// TIA Portal V20 export
FUNCTION "E001" : Void   // FC2, FBD
{ S7_Optimized_Access := 'TRUE' }
// stored: SetENOAutomatically false
   VAR_TEMP
      Stirrer_TimeMs : DInt;
      State : "Service_States";
   END_VAR
BEGIN

REGION Network 1: Channel input
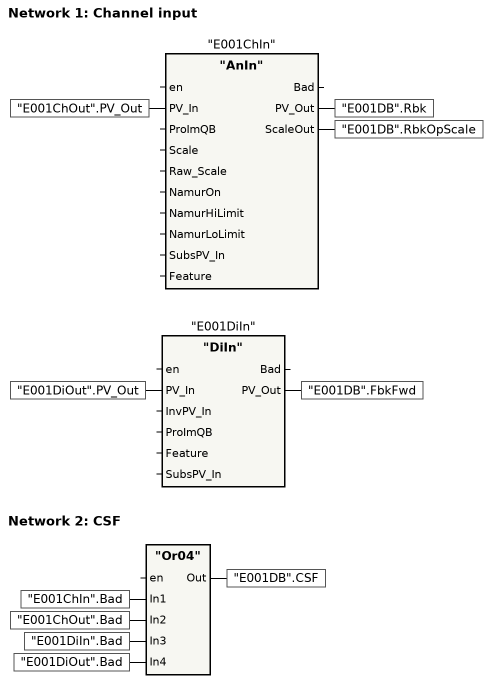
   "E001ChIn"(PV_In := "E001ChOut".PV_Out, PV_Out => "E001DB".Rbk, ScaleOut => "E001DB".RbkOpScale);   // "AnIn"
   "E001DiIn"(PV_In := "E001DiOut".PV_Out, PV_Out => "E001DB".FbkFwd);   // "DiIn"
END_REGION

REGION Network 2: CSF
   "Or04"(In1 := "E001ChIn".Bad,
          In2 := "E001ChOut".Bad,
          In3 := "E001DiIn".Bad,
          In4 := "E001DiOut".Bad,
          Out => "E001DB".CSF);
END_REGION

REGION Network 3: Interlock
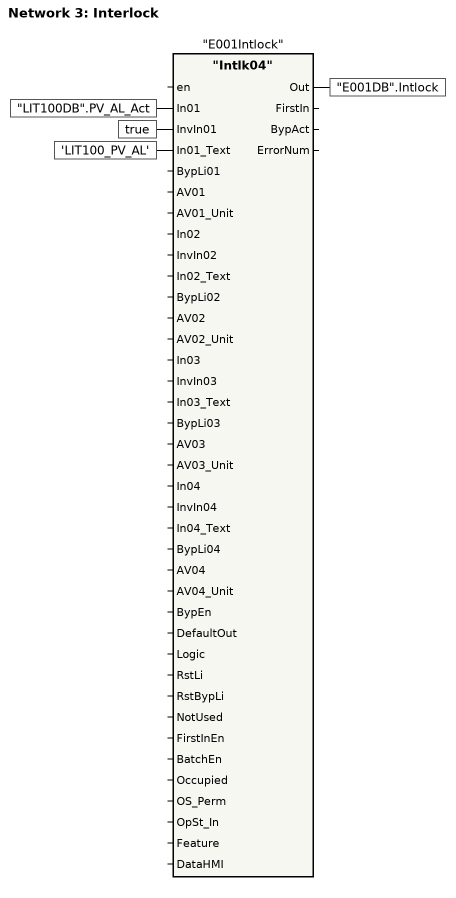
   "E001Intlock"(In01 := "LIT100DB".PV_AL_Act,   // "Intlk04"
                 InvIn01 := true,
                 In01_Text := 'LIT100_PV_AL',
                 Out => "E001DB".Intlock);
END_REGION

REGION Network 4: MotSpdCL
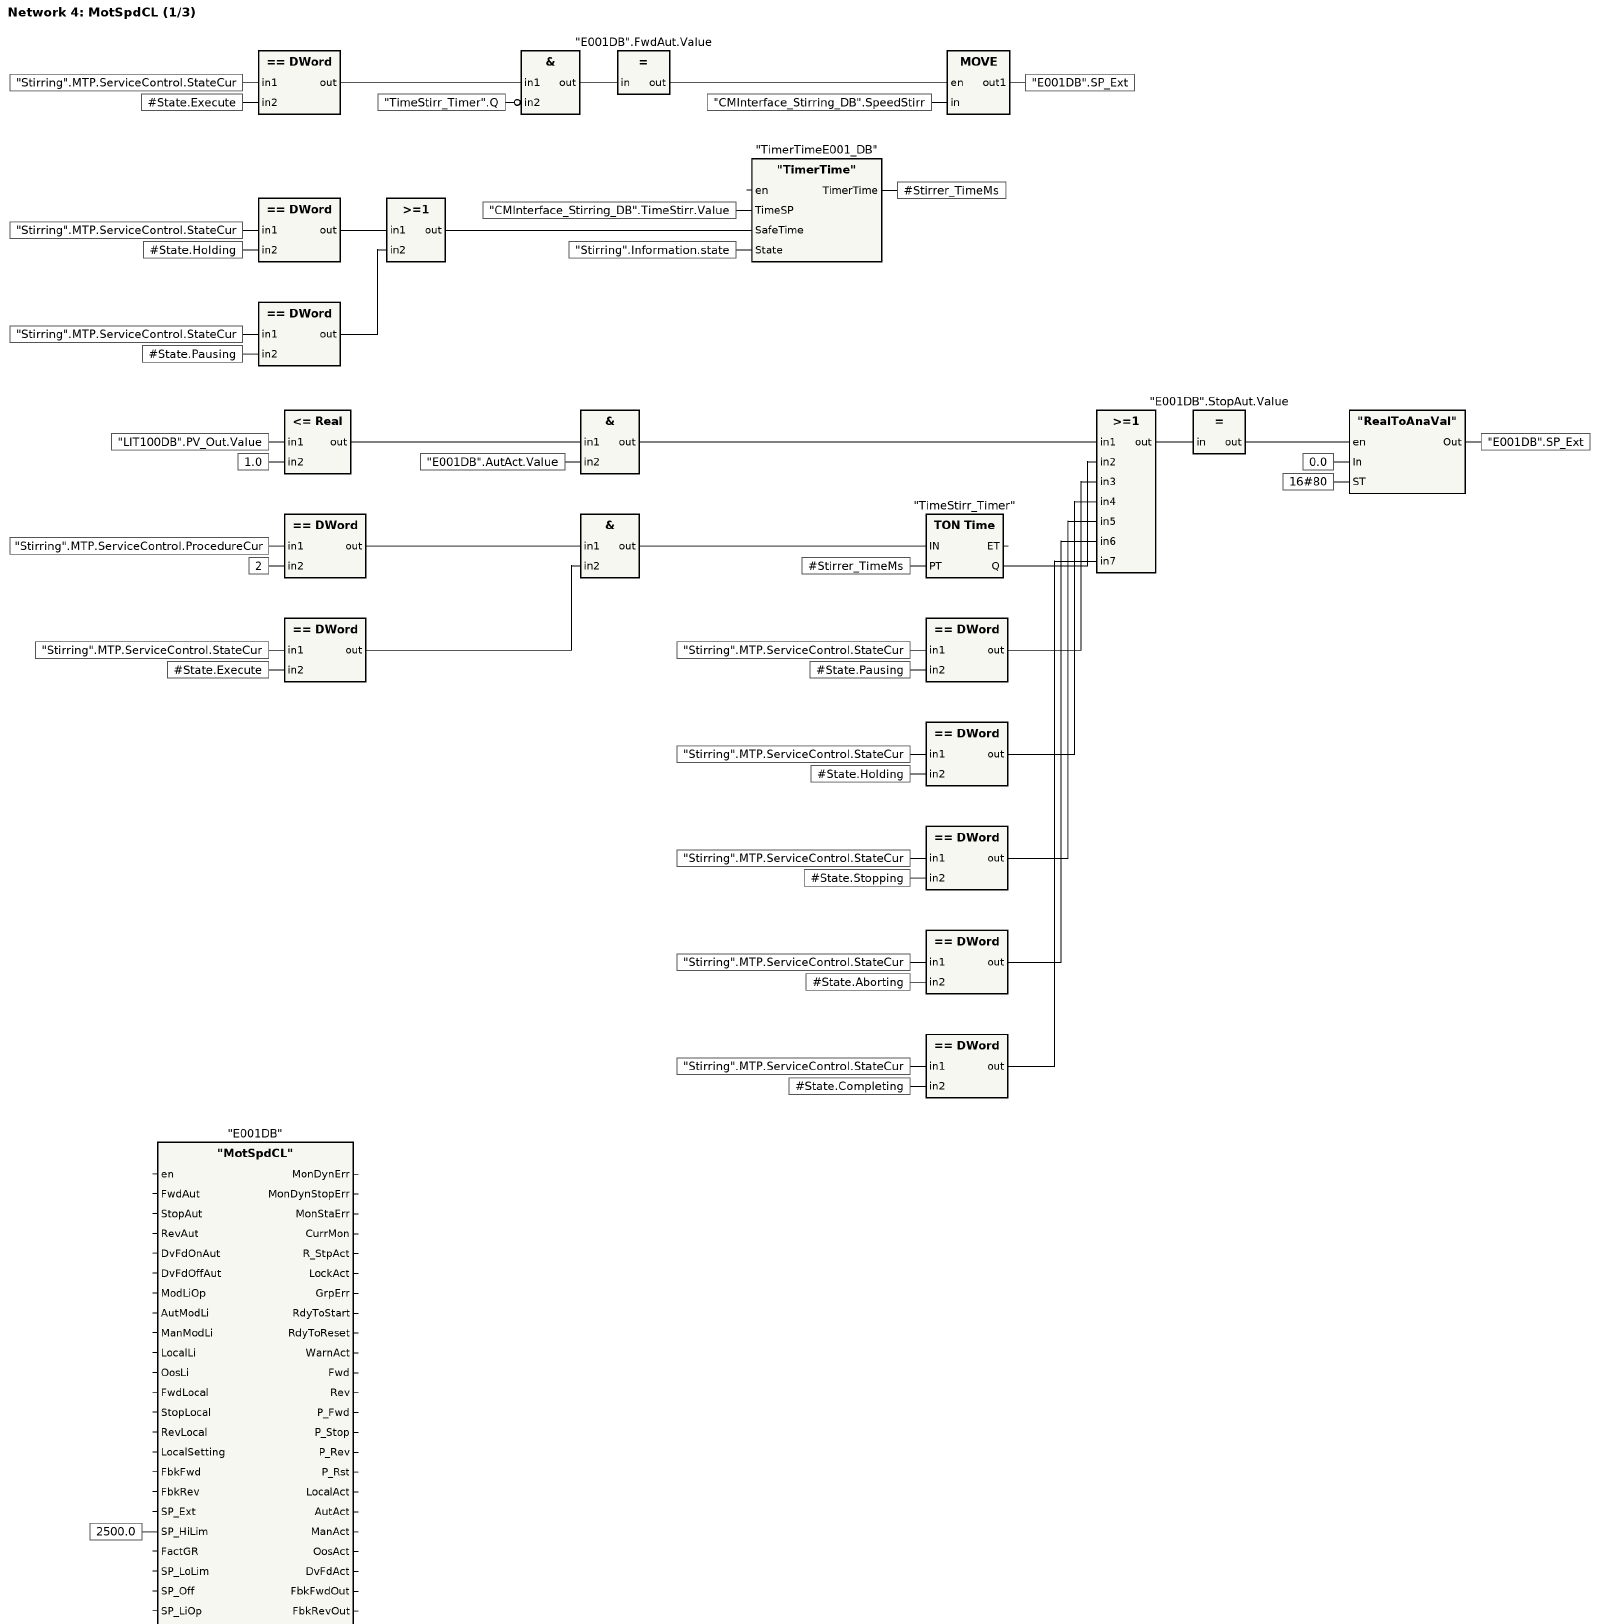
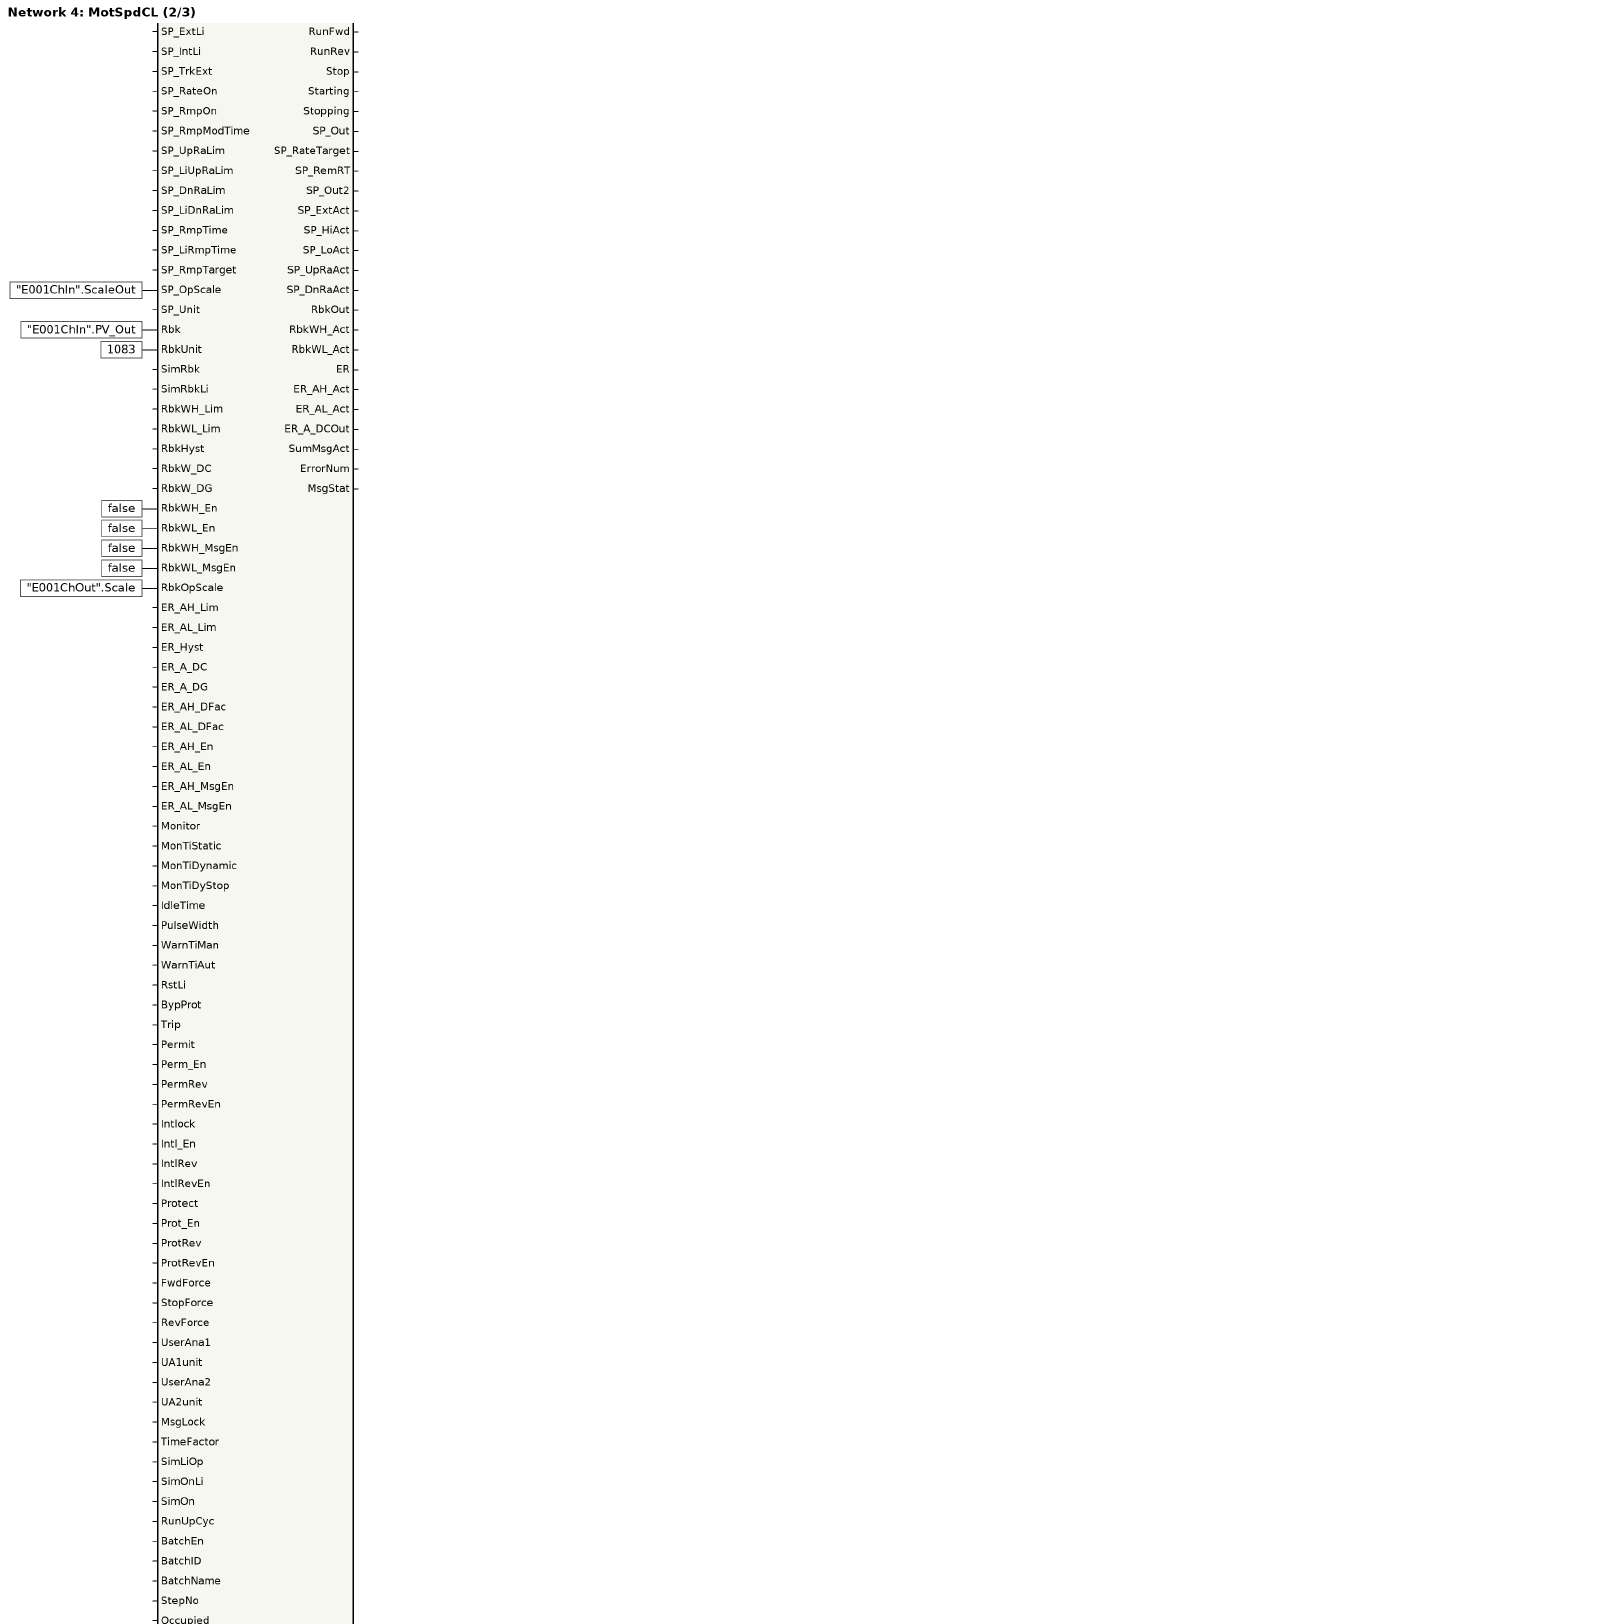
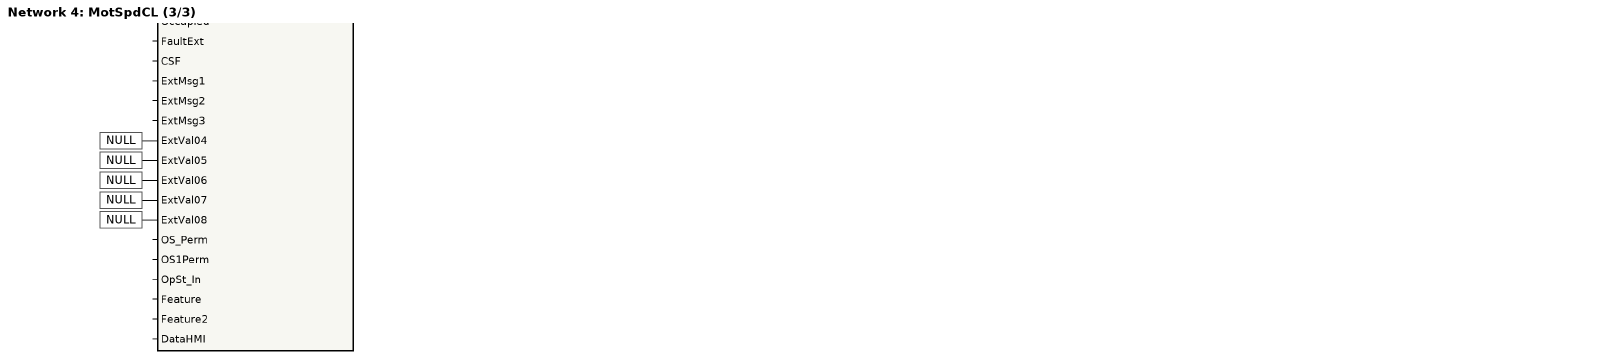
   "E001DB".FwdAut.Value := ("Stirring".MTP.ServiceControl.StateCur = #State.Execute) AND NOT "TimeStirr_Timer".Q;
   IF "E001DB".FwdAut.Value THEN "E001DB".SP_Ext := "CMInterface_Stirring_DB".SpeedStirr; END_IF;
   "TimerTimeE001_DB"(TimeSP := "CMInterface_Stirring_DB".TimeStirr.Value,   // "TimerTime"
                      SafeTime := ("Stirring".MTP.ServiceControl.StateCur = #State.Holding) OR ("Stirring".MTP.ServiceControl.StateCur = #State.Pausing),
                      State := "Stirring".Information.state,
                      TimerTime => #Stirrer_TimeMs);
   "TimeStirr_Timer".TON(IN := ("Stirring".MTP.ServiceControl.ProcedureCur = 2) AND ("Stirring".MTP.ServiceControl.StateCur = #State.Execute),
                         PT := #Stirrer_TimeMs);
   "E001DB".StopAut.Value := (("LIT100DB".PV_Out.Value <= 1.0) AND "E001DB".AutAct.Value) OR "TimeStirr_Timer".Q OR ("Stirring".MTP.ServiceControl.StateCur = #State.Pausing) OR ("Stirring".MTP.ServiceControl.StateCur = #State.Holding) OR ("Stirring".MTP.ServiceControl.StateCur = #State.Stopping) OR ("Stirring".MTP.ServiceControl.StateCur = #State.Aborting) OR ("Stirring".MTP.ServiceControl.StateCur = #State.Completing);
   IF "E001DB".StopAut.Value THEN "RealToAnaVal"(In := 0.0, ST := 16#80, Out => "E001DB".SP_Ext); END_IF;
   "E001DB"(SP_HiLim := 2500.0,   // "MotSpdCL"
            SP_OpScale := "E001ChIn".ScaleOut,
            Rbk := "E001ChIn".PV_Out,
            RbkUnit := 1083,
            RbkWH_En := false,
            RbkWL_En := false,
            RbkWH_MsgEn := false,
            RbkWL_MsgEn := false,
            RbkOpScale := "E001ChOut".Scale,
            ExtVal04 := NULL,
            ExtVal05 := NULL,
            ExtVal06 := NULL,
            ExtVal07 := NULL,
            ExtVal08 := NULL);
END_REGION

REGION Network 5: MTP
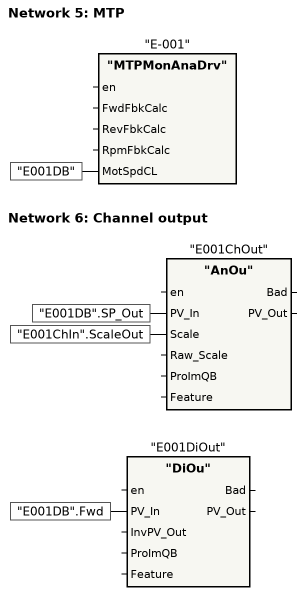
   "E-001"(MotSpdCL := "E001DB");   // "MTPMonAnaDrv"
END_REGION

REGION Network 6: Channel output
   "E001ChOut"(PV_In := "E001DB".SP_Out, Scale := "E001ChIn".ScaleOut);   // "AnOu"
   "E001DiOut"(PV_In := "E001DB".Fwd);   // "DiOu"
END_REGION
END_FUNCTION
